{attribute 'qualified_only'}
{attribute 'strict'}
TYPE VerkeerslichtStatus :
(
	Rood := 0,    // 0
    Geel := 1,    // 1
    Groen := 2    // 2
);
END_TYPE

(* stored: Version 1.1.0.1, ProductVersion 3.1.4024.12
   EnumerationTextList VerkeerslichtStatus: Id {600c2b9a-6474-44a7-a0f0-374db7846edb} *)
